// TIA Portal V20 export
FUNCTION "SysCheckSafetyModule" : Void   // FC2157, FBD
TITLE = SysCheckSafetyModules
{ S7_Optimized_Access := 'TRUE' }
// stored: AutoNumber false, SetENOAutomatically false
   VAR_INPUT
      AdrET : HW_DEVICE;   // Address of the ET station
      AdrMO_Start : HW_IO;   // Address of first ET modul
      AdrMO_End : HW_IO;   // Address of last ET modul
   END_VAR
   VAR_OUTPUT
      ErrThis : Bool;
   END_VAR
   VAR_TEMP
      i : Int;
      tFirstSlot : Int;
      tLastSlot : Int;
      t_Err : Bool;
      t_RetVal : Int;
      tState : Array[0..127] of Bool;
      tGeoAddr : GEOADDR;
   END_VAR
   VAR_TEMP   // added for the SCL form of the ladder/FBD networks
      _w1 : Bool;
      _w2 : Bool;
   END_VAR
BEGIN

REGION Network 1: read module slot numbers
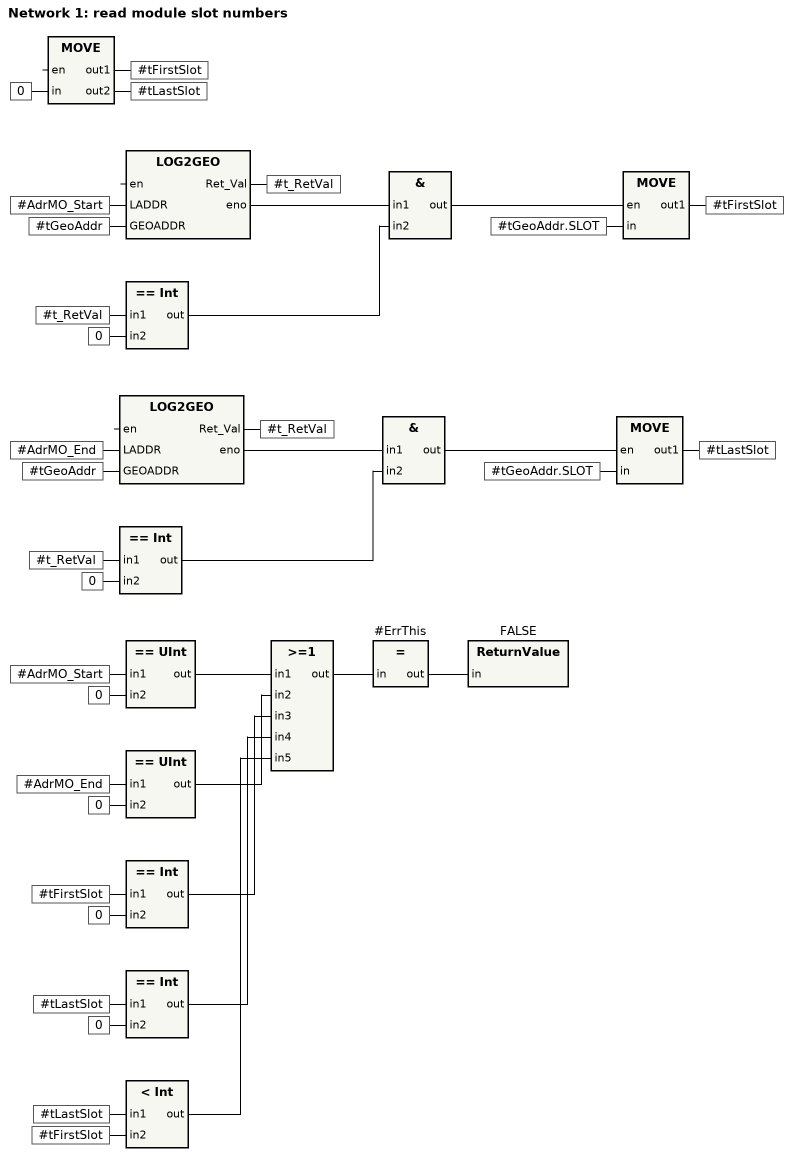
   #tFirstSlot := 0;
   #tLastSlot := 0;
   #t_RetVal := LOG2GEO(LADDR := #AdrMO_Start, GEOADDR := #tGeoAddr, ENO => #_w1);
   IF #_w1 AND (#t_RetVal = 0) THEN #tFirstSlot := #tGeoAddr.SLOT; END_IF;
   #t_RetVal := LOG2GEO(LADDR := #AdrMO_End, GEOADDR := #tGeoAddr, ENO => #_w2);
   IF #_w2 AND (#t_RetVal = 0) THEN #tLastSlot := #tGeoAddr.SLOT; END_IF;
   #ErrThis := (#AdrMO_Start = 0) OR (#AdrMO_End = 0) OR (#tFirstSlot = 0) OR (#tLastSlot = 0) OR (#tLastSlot < #tFirstSlot);
   IF #ErrThis THEN
       ENO := FALSE;
       RETURN;
   END_IF;
END_REGION

REGION Network 2: read station status
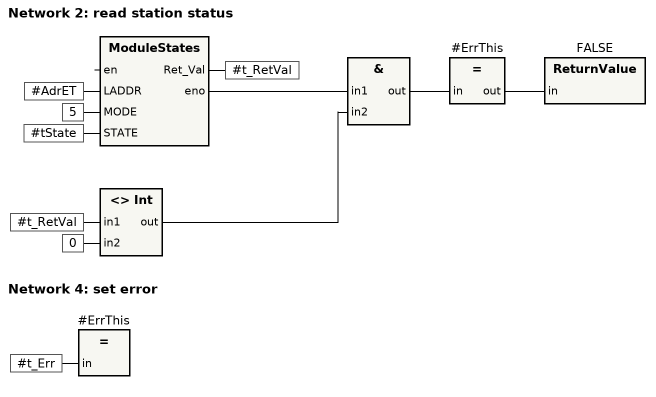
   #t_RetVal := ModuleStates(LADDR := #AdrET, MODE := 5, STATE := #tState, ENO => #_w1);
   #ErrThis := #_w1 AND (#t_RetVal <> 0);
   IF #ErrThis THEN
       ENO := FALSE;
       RETURN;
   END_IF;
END_REGION

REGION Network 3 (SCL): search for fault
   #t_Err := false;
   FOR #i := #tFirstSlot TO #tLastSlot DO
       IF #tState[#i+1] THEN
           #t_Err := true;
           EXIT;
       END_IF;
   END_FOR;
END_REGION

REGION Network 4: set error
   #ErrThis := #t_Err;
END_REGION
END_FUNCTION
